// TIA Portal V17 export
// export: Created 2022-03-29T18:52:11.6299411Z, ExportSetting WithDefaults, DisplayName Totally Integrated Automation Portal, DisplayVersion V17, DisplayName TIA Portal Openness, DisplayVersion V17, DisplayName TIA Portal Version Control Interface, DisplayVersion V17, DisplayName STEP 7 Professional, DisplayVersion V17, DisplayName STEP 7 Safety, DisplayVersion V17, DisplayName WinCC Advanced / Unified PC, DisplayVersion V17
FUNCTION_BLOCK "EM00_CM03_ConveyorCrossing"   // FB31653, LAD
TITLE = EM00_CM03
{ S7_Optimized_Access := 'TRUE' }
AUTHOR : tech.team.motioncontrol@siemens.com
FAMILY : CPG
VERSION : 1.1
// Support: tech.team.motioncontrol@siemens.com
// stored: AutoNumber true, IsIECCheckEnabled false, IsRetainMemResEnabled false, MemoryReserve 100, SetENOAutomatically false, UDAEnableTagReadback false
   VAR
      statDummyBool { ExternalAccessible := 'False'; ExternalVisible := 'False'; ExternalWritable := 'False'} : Bool;   // dummy bool - placeholder
      instConveyorCrossing { S7_SetPoint := 'True'} : "ConveyorCrossing";
   END_VAR
BEGIN

REGION Network 1: *** Begin the Setpoint Management Information Section ***
END_REGION

REGION Network 2: *** Begin the Logic Section ***
END_REGION

REGION Network 3: Conveyor crossing instance
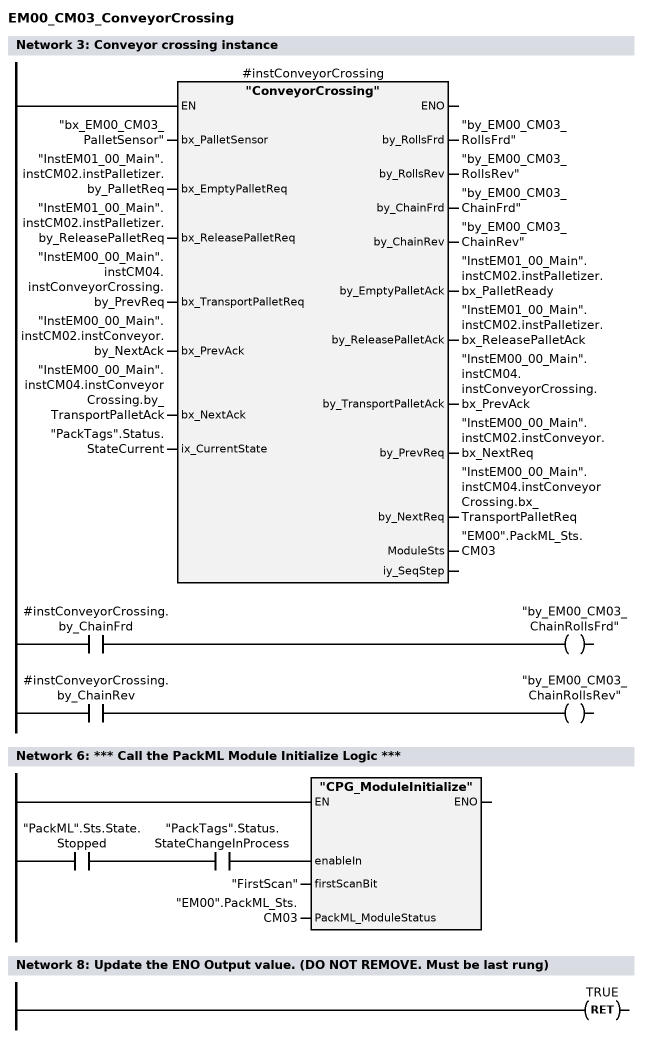
   RUNG wire#powerrail
      #instConveyorCrossing(bx_PalletSensor := "bx_EM00_CM03_PalletSensor", bx_EmptyPalletReq := "InstEM01_00_Main".instCM02.instPalletizer.by_PalletReq, bx_ReleasePalletReq := "InstEM01_00_Main".instCM02.instPalletizer.by_ReleasePalletReq, bx_TransportPalletReq := "InstEM00_00_Main".instCM04.instConveyorCrossing.by_PrevReq, bx_PrevAck := "InstEM00_00_Main".instCM02.instConveyor.by_NextAck, bx_NextAck := "InstEM00_00_Main".instCM04.instConveyorCrossing.by_TransportPalletAck, ix_CurrentState := "PackTags".Status.StateCurrent, by_RollsFrd => "by_EM00_CM03_RollsFrd", by_RollsRev => "by_EM00_CM03_RollsRev", by_ChainFrd => "by_EM00_CM03_ChainFrd", by_ChainRev => "by_EM00_CM03_ChainRev", by_EmptyPalletAck => "InstEM01_00_Main".instCM02.instPalletizer.bx_PalletReady, by_ReleasePalletAck => "InstEM01_00_Main".instCM02.instPalletizer.bx_ReleasePalletAck, by_TransportPalletAck => "InstEM00_00_Main".instCM04.instConveyorCrossing.bx_PrevAck, by_PrevReq => "InstEM00_00_Main".instCM02.instConveyor.bx_NextReq, by_NextReq => "InstEM00_00_Main".instCM04.instConveyorCrossing.bx_TransportPalletReq, ModuleSts => "EM00".PackML_Sts.CM03, iy_SeqStep =>)
   END_RUNG
   RUNG wire#powerrail
      Contact( #instConveyorCrossing.by_ChainFrd )
      Coil( "by_EM00_CM03_ChainRollsFrd" )
   END_RUNG
   RUNG wire#powerrail
      Contact( #instConveyorCrossing.by_ChainRev )
      Coil( "by_EM00_CM03_ChainRollsRev" )
   END_RUNG
   // the same network as SCL:
   #instConveyorCrossing(bx_PalletSensor := "bx_EM00_CM03_PalletSensor",   // "ConveyorCrossing"
                         bx_EmptyPalletReq := "InstEM01_00_Main".instCM02.instPalletizer.by_PalletReq,
                         bx_ReleasePalletReq := "InstEM01_00_Main".instCM02.instPalletizer.by_ReleasePalletReq,
                         bx_TransportPalletReq := "InstEM00_00_Main".instCM04.instConveyorCrossing.by_PrevReq,
                         bx_PrevAck := "InstEM00_00_Main".instCM02.instConveyor.by_NextAck,
                         bx_NextAck := "InstEM00_00_Main".instCM04.instConveyorCrossing.by_TransportPalletAck,
                         ix_CurrentState := "PackTags".Status.StateCurrent,
                         by_RollsFrd => "by_EM00_CM03_RollsFrd",
                         by_RollsRev => "by_EM00_CM03_RollsRev",
                         by_ChainFrd => "by_EM00_CM03_ChainFrd",
                         by_ChainRev => "by_EM00_CM03_ChainRev",
                         by_EmptyPalletAck => "InstEM01_00_Main".instCM02.instPalletizer.bx_PalletReady,
                         by_ReleasePalletAck => "InstEM01_00_Main".instCM02.instPalletizer.bx_ReleasePalletAck,
                         by_TransportPalletAck => "InstEM00_00_Main".instCM04.instConveyorCrossing.bx_PrevAck,
                         by_PrevReq => "InstEM00_00_Main".instCM02.instConveyor.bx_NextReq,
                         by_NextReq => "InstEM00_00_Main".instCM04.instConveyorCrossing.bx_TransportPalletReq,
                         ModuleSts => "EM00".PackML_Sts.CM03);
   "by_EM00_CM03_ChainRollsFrd" := #instConveyorCrossing.by_ChainFrd;
   "by_EM00_CM03_ChainRollsRev" := #instConveyorCrossing.by_ChainRev;
END_REGION

REGION Network 4: *** Begin the Event Information Section ***
END_REGION

REGION Network 5: *** Begin the State Model Status Feedback Section ***
END_REGION

REGION Network 6: *** Call the PackML Module Initialize Logic ***
   RUNG wire#powerrail
      "CPG_ModuleInitialize"(enableIn := wire#w1, firstScanBit := "FirstScan", PackML_ModuleStatus := "EM00".PackML_Sts.CM03)
   END_RUNG
   RUNG wire#powerrail
      Contact( "PackML".Sts.State.Stopped )
      Contact( "PackTags".Status.StateChangeInProcess )
   END_RUNG wire#w1
   // the same network as SCL:
   "CPG_ModuleInitialize"(enableIn := "PackML".Sts.State.Stopped AND "PackTags".Status.StateChangeInProcess,
                          firstScanBit := "FirstScan",
                          PackML_ModuleStatus := "EM00".PackML_Sts.CM03);
END_REGION

REGION Network 8: Update the ENO Output value. (DO NOT REMOVE. Must be last rung)
   RUNG wire#powerrail
      ReturnCoil( TRUE )
   END_RUNG
   // the same network as SCL:
   ENO := TRUE;
   RETURN;
END_REGION
END_FUNCTION_BLOCK
